(* CODESYS project ExampleProject 1.0.0.0.project

Project tree, tasks and I/O mapping:
  CODESYS_Control_for_Raspberry_Pi_SL : CODESYS Control for Raspberry Pi SL, 3S - Smart Software Solutions GmbH, version 3.5.12.0
    application Application
      libraries: Util, * (System)
      task Task (cyclic, interval t#50ms, priority 1, watchdog 100 ms x 1) calls PRG_Monarco_HAT_Examples
      task VISU_TASK (cyclic, interval 100 ms, priority 31) calls VisuElems.Visu_Prg
      program PRG_Monarco_HAT_Examples [ST]
      RS485/
        Enums/
          data type SERIAL_LINE_MODE
        FB/
          function block SERIAL_LINE [ST]: Fb_init, CLOSE
        Visualisation/
          visualisation Visualisation
          visualisation SERIAL_LINE_VISU
    SoftMotion General Axis Pool
    I²C
    SPI
      SPI_master : SPI master, 3S - Smart Software Solutions GmbH, version 1.0.0.0
          settings: _diBitsPerWord = 8; _diMaxSpeed = 1000000
        Monarco_HAT : Monarco HAT, Monarco.io, version 1.0.0.0
    GPIOs_A_B : GPIOs B+/Pi2, 3S - Smart Software Solutions GmbH, version 3.5.11.0
        unmapped channels: digital inputs (GPIO0..GPIO31), digital outputs (GPIO0..GPIO31)
    Onewire
    Camera device
      <Empty>
  libraries: Raspberry Pi Peripherals, 3.5.11.0 (3S - Smart Software Solutions GmbH); IoStandard, * (System); CAA Types Extern, * (CAA Technical Workgroup); Standard, * (System); SysTypes Interfaces, * (System); CAA Memory, * (CAA Technical Workgroup); Component Manager, * (System); CmpLog, * (System); CmpErrors Interfaces, * (System); CAA SerialCom, * (CAA Technical Workgroup); CAA Real Time Clock Extern, * (CAA Technical Workgroup); VisuSymbols, 3.5.10.0 (System)
  text list GlobalTextList
*)

// CODESYS_Control_for_Raspberry_Pi_SL/Application/RS485/Enums/SERIAL_LINE_MODE
TYPE SERIAL_LINE_MODE : (SL_READ, SL_WRITE, SL_READWRITE);
END_TYPE

// CODESYS_Control_for_Raspberry_Pi_SL/Application/PRG_Monarco_HAT_Examples
PROGRAM PRG_Monarco_HAT_Examples
VAR
	xOPm 			: BOOL := FALSE;// is the SPI master operational?
	xOPs			: BOOL := FALSE;// is the SPI slave operational?
	xExecute		: BOOL := TRUE;
	I				: INT;
	LedValue		: BYTE;	

	uiWDTime 		: UINT := 123;
	uiNewWDTime		: UINT := 500;
	xSetWd			: BOOL := FALSE;
	xWrite			: BOOL;
	DOut			: MNR.stDOut;
	DIn				: MNR.stDIn;
	AOut			: MNR.stAOut;     		
	AIn				: MNR.stAIn;	
	K	 			: INT;
	
	HatInfo			: MNR.stHATinfo;
	
	xSetHwConfig1	: BOOL;
	xGetHwConfig1	: BOOL;
	xTerminated		: BOOL;
	xAIN1shunt		: BOOL;
	xAIN2shunt		: BOOL;
	myHWConfig1		: MNR.stHWConfig1;
	curHWConfig1	: MNR.stHWConfig1;
	
	Blink			: UTIL.BLINK;
	GetDateAndTime	: RTCLK.GetDateAndTime;
	xEnablePWM		: BOOL;
	xDone			: BOOL;
	xBusy			: BOOL;
	xError			: BOOL;
	eError			: RTCLK.ERROR;
	eTimezone		: RTCLK.PERIODE;
	VarTimeCur		: DATE_AND_TIME;
	
	xSetConfig		: BOOL;
	xGetConfig		: BOOL;
	eMode			: MNR.eCounterMode 			:= MNR.eCounterMode.Off;
	eDirection		: MNR.eCounterDirection 	:= MNR.eCounterDirection.Up;
	eActiveEdge		: MNR.eCounterActiveEdge	:= MNR.eCounterActiveEdge.Rising;
	eCapture		: MNR.eCounterCapture		:= MNR.eCounterCapture.Disabled;
	myConfig1 		: MNR.stCounter1Config;
	getConfig1		: MNR.stCounter1Config;
	
	xTwoLinesOld	: BOOL;
	FirstSerialLine	: SERIAL_LINE;	
	uiCurBaudrate	: UINT;	
	xGetBaudrate	: BOOL := TRUE;
	xSetBaudrate	: BOOL;           	
	xSetMode		: BOOL;
	xGetMode		: BOOL;
	xSetRS485Mode	: BOOL;
	xGetRS485Mode	: BOOL;
	eDatabits		: MNR.eRS485Databits 	:= MNR.eRS485Databits.eight;
	eParity			: MNR.eRS485Parity 		:= MNR.eRS485Parity.none;
	eStopbits		: MNR.eRS485Stopbits 	:= MNR.eRS485Stopbits.One;
	ServiceResponse : MNR.stServiceResponse;
	myMode 			: MNR.stRS485Mode;
	xGetHOSTBaudrate: BOOL := TRUE;
	uiHOSTBaudrate	: UINT;
END_VAR

(*============================== VARIOUS HAT DEMONSTRATION USAGE EXAMPLES ==============================
	Wiring for Monarco self test;
	Wire all AO channels to the AI channels (2 AO, 2 AI),
	Wire all DO channels to the DI channels (4 DO, 4 DI),
	Wire the GND to DIn COM-,
	Wire RS485 Rx to Tx,
	Ready!
*)
xOPm  := SPI_Master.Operational;
xOPs  := Monarco_HAT.Operational;
HatInfo	:= Monarco_HAT.HATinfo;


(*============================== Monarco Leds  ==============================*)
IF I <= 7 THEN
	I := I + 1;
ELSE
	I := 0;
END_IF
LEDValue 			:= TO_BYTE( EXPT(2,I) );
Monarco_HAT.SetUserLED( byLeds := LEDValue);


(*============================== Watchdog  ==============================*)
uiWDTime    := Monarco_HAT.Watchdog;
IF xSetWd THEN
	// set
	Monarco_HAT.Watchdog := uiNewWDTime;
	xSetWd	:= FALSE;
END_IF


(*============================== Monarco DO as a struct  ==============================*)
K := K + 1;
IF K > 4 THEN
	K := 0;
END_IF;
DOut.xDOut1 := (K=1);
DOut.xDOut2 := (K=2);
DOut.xDOut3 := (K=3);
DOut.xDOut4 := (K=4);
Monarco_HAT.setDOut( stDOut := Dout);
/// two "overloads" are available;
//Monarco_HAT.setDOutBool 
//Monarco_HAT.setDOutByte

(*============================== Monarco DI as a struct  ==============================*)
Monarco_HAT.getDIn( stDIn => DIn );
///two "overloads" are available;
//Monarco_HAT.getDInBool
//Monarco_HAT.getDInByte


(*============================== Monarco AO as a struct  ==============================*)
AOut.wAOut1 := AOut.wAOut1 + 1;
IF AOut.wAOut1 >4095 THEN
	AOut.wAOut1 := 0;
END_IF
AOut.wAOut2 := AOut.wAOut1;
Monarco_HAT.setAOut( stAOut := AOut );
/// One "overload" is available;
//Monarco_Hat.setAOutWord


(*============================== AI as a struct  ==============================*)
Monarco_HAT.getAIn( stAIn => AIn);
/// One "overload" is available;
//Monarco_Hat.getAInWord


(*============================== HWCONFIG ==============================*)
// read current config
IF xGetHwConfig1 THEN
	curHWConfig1 := Monarco_HAT.HWConfig1;
	xGetHwConfig1 := FALSE;
END_IF

IF xSetHwConfig1 THEN
	myHWConfig1.xTerminated := xTerminated;
	myHWConfig1.xAIn1shunt  := xAIN1shunt;
	myHWConfig1.xAIN2shunt  := xAIN2shunt;
	// set new config
	Monarco_HAT.HWConfig1 := myHWConfig1;
	// read current config
	xGetHwConfig1 := TRUE;
	xSetHwConfig1 := FALSE;
END_IF


(*============================== One Wire ==============================*)
// One Wire is ready to use after the HAT overlay is installed
// A usage example is not provided

(*============================== RTC ==============================*)
// RTC is ready to use after the HAT overlay is installed
Blink( ENABLE := TRUE, TIMELOW := T#500MS, TIMEHIGH := T#500MS);
GetDateAndTime(
	xExecute:= Blink.OUT, // pulse for actual time
	xDone=> xDone, 
	xBusy=> xBusy, 
	xError=> xError, 
	eError=> eError, 
	eTimezone=> eTimezone);
IF xDone AND NOT xError THEN
	VarTimeCur := GetDateAndTime.dtDateAndTime;
END_IF


(*============================== COUNTER ==============================*)
// Setting an arbitrairy mode via property
myConfig1.eMode			:= eMode;
myConfig1.eDirection	:= eDirection;
myConfig1.eActiveEdge	:= eActiveEdge;
IF xSetConfig THEN
	Monarco_HAT.Counter1Config := myConfig1;
	xSetConfig := FALSE;
END_IF
IF xGetConfig THEN
	getConfig1 := Monarco_HAT.Counter1Config;
	xGetConfig := FALSE;
END_IF


(*============================== PWM ==============================*)
Monarco_HAT.setPWM1freq( udiHz := 5000); // 5000Hz
Monarco_HAT.setPWM2freq( udiHz := 100); // 100Hz
IF xEnablePWM THEN
	Monarco_HAT.setDutyCycleDOut1(rDutyCycle := 0.04); //4%
	Monarco_HAT.setDutyCycleDOut2(rDutyCycle := 0.20); //20%
	Monarco_HAT.setDutyCycleDOut3(rDutyCycle := 0.45); //45%
	Monarco_HAT.setDutyCycleDOut4(rDutyCycle := 0.75); //75%
ELSE
	/// Disable the PWM
	Monarco_HAT.setDutyCycleDOut1(rDutyCycle := 0.0); //0%
	Monarco_HAT.setDutyCycleDOut2(rDutyCycle := 0.0); //0%
	Monarco_HAT.setDutyCycleDOut3(rDutyCycle := 0.0); //0%
	Monarco_HAT.setDutyCycleDOut4(rDutyCycle := 0.0); //0%
END_IF


(*============================== Counters ==============================*)
// Counters are ready to use after the HAT overlay is installed
// A usage example is not provided


(*============================== RS485 ==============================*)
//// Adapt the enums for COM library interoperability, in this case Monarco.IO to CAA_COM_LIB;
//CASE getMode.Databits OF
//	MNR.eRS485Databits.Five			: udiByteSize := 5;
//	MNR.eRS485Databits.Six			: udiByteSize := 6;
//	MNR.eRS485Databits.Seven		: udiByteSize := 7;
//	MNR.eRS485Databits.Eight		: udiByteSize := 8;
//END_CASE
//CASE getMode.Parity OF
//	MNR.eRS485Parity.Even			: paParity := COM.PARITY.EVEN;
//	MNR.eRS485Parity.Odd			: paParity := COM.PARITY.ODD;
//	MNR.eRS485Parity.None			: paParity := COM.PARITY.None;
//END_CASE
//CASE getMode.Stopbits OF
//	MNR.eRS485STOPBITS.One			: sbStopBits := COM.STOPBIT.ONESTOPBIT;	
//	MNR.eRS485STOPBITS.OneAndAHalf	: sbStopBits := COM.STOPBIT.ONE5STOPBITS;	
//	MNR.eRS485STOPBITS.Two			: sbStopBits := COM.STOPBIT.TWOSTOPBITS;
//ELSE
//// 1/2 stopbit *not* supported in CAA COM lib!
//	MNR.eRS485STOPBITS.Half			: sbStopBits := COM.STOPBIT.ONESTOPBIT;
//END_CASE

IF xGetBaudrate THEN
	uiCurBaudrate := Monarco_HAT.RS485Baudrate;
	xGetBaudrate := FALSE;
END_IF
IF xSetBaudrate THEN
	// set 320000 baud 
	Monarco_HAT.RS485Baudrate := 320;
	xSetBaudrate := FALSE;
END_IF
// Setting the mode via a service request
IF xSetMode THEN
	// Setting 8,E,1 (Default 8,N,1)
	Monarco_HAT.serviceRequest( wValue := 16#0039, eCommand := MNR.eServiceCommand.SDC_FIXED_RS485MODE, xWrite := TRUE);
	xSetMode := FALSE;
END_IF
// Reading HOST UART mode via a service request
IF xGetMode THEN
	Monarco_HAT.serviceRequest( wValue := MNR.ParamList.MONARCO_SERVICE_STATUS_OK, eCommand := MNR.eServiceCommand.SDC_FIXED_HOST_UART, xWrite := FALSE);
	xGetMode := FALSE;
	// Read last response, default will be 16#0038 (8,N,1)
	// When setmode this will yield 16#0039
	Monarco_HAT.getServiceResponse(Response => ServiceResponse);
END_IF
// Setting an arbitrairy mode via property
myMode.eDatabits	:= eDatabits;
myMode.eParity		:= eParity;
myMode.eStopbits	:= eStopbits;
IF xSetRS485Mode THEN
	Monarco_HAT.RS485Mode := myMode;
	xSetRS485Mode := FALSE;
END_IF
IF xGetRS485Mode THEN
	myMode := Monarco_HAT.RS485Mode;
	xGetRS485Mode := FALSE;
END_IF
// should be 115200
IF xGetHOSTBaudrate THEN
 	uiHostBaudrate := Monarco_HAT.HostBaudrate;
	xGetHOSTBaudrate := FALSE;
END_IF;

// Sourcecode is included in this project under a separate RS485 section
FirstSerialLine(
		slMode:= SL_READWRITE, 
		udiPort:= 1, 							
		udiBaudrate:= 115200,
		paParity:= COM.PARITY.NONE,
		sbStopBits:= COM.STOPBIT.ONESTOPBIT,
		udiByteSize := 8);

END_PROGRAM

// CODESYS_Control_for_Raspberry_Pi_SL/Application/RS485/FB/SERIAL_LINE
FUNCTION_BLOCK SERIAL_LINE
VAR_INPUT
	slMode				: SERIAL_LINE_MODE;
	udiPort				: UDINT;
	udiBaudrate			: UDINT;
	sbStopBits			: COM.STOPBIT:= COM.STOPBIT.ONESTOPBIT;
	paParity			: COM.PARITY:= COM.PARITY.EVEN;
	sWriteText			: STRING:= 'Hello Raspberry and Monarco! ';
	udiByteSize			: UDINT;
END_VAR
VAR_OUTPUT
	sReadText			: STRING;
	errError			: COM.ERROR;
	xReadSuccess		: BOOL;
	xWriteSuccess		: BOOL;
	xClosed				: BOOL:= TRUE;
END_VAR
VAR
	iState				: INT;
	tTimer				: TON;
	comOpen				: COM.Open; (* Instance of the function block for opening a port *)
	hCom				: CAA.HANDLE; (* handle of the port*)
	aParameter			: ARRAY [1..7] OF COM.PARAMETER;
	comWrite			: COM.Write;	(* Instance of the Write function  block *)
	bWriteBuffer		: ARRAY [1..80] OF BYTE; (*Used to write data to the serial port*)
	szWrite				: CAA.SIZE;
	comRead				: COM.Read; (* Instance of the Read function block *)
	bReadBuffer			: ARRAY [1..80] OF BYTE; (*Used to read data from the serial port*)
	szRead				: CAA.SIZE;
	comClose			: COM.Close; (* Instance of the function block for closing a port *)
END_VAR

CASE iState OF
	
	0:	// The parameter for the COM Ports are set
		aParameter[1].udiParameterId:= COM.CAA_Parameter_Constants.udiPort;
		aParameter[1].udiValue:= udiPort;
		aParameter[2].udiParameterId:= COM.CAA_Parameter_Constants.udiBaudrate;
		aParameter[2].udiValue:= udiBaudrate;		
		aParameter[3].udiParameterId:= COM.CAA_Parameter_Constants.udiStopBits;
		aParameter[3].udiValue:= sbStopBits;
		aParameter[4].udiParameterId:= COM.CAA_Parameter_Constants.udiParity;
		aParameter[4].udiValue:= paParity;
		aParameter[5].udiParameterId:= COM.CAA_Parameter_Constants.udiTimeout;
		aParameter[5].udiValue:= 0;
		aParameter[6].udiParameterId:= COM.CAA_Parameter_Constants.udiBinary;
		aParameter[6].udiValue:= 0;
		aParameter[7].udiParameterId:= COM.CAA_Parameter_Constants.udiByteSize;
		aParameter[7].udiValue:= udiByteSize;
		
		iState:= 1;
		
	1:	//First the COM Port is opened
		comOpen(xExecute:= TRUE, usiListLength:= SIZEOF(aParameter) / SIZEOF(COM.PARAMETER), pParameterList:= ADR(aParameter), hCom=> hCom);
		xClosed:= FALSE;
		IF comOpen.xDone THEN
			comOpen(xExecute:= FALSE);
			//depending on the mode the state for reading or writing is set
			IF slMode = SL_READ OR slMode = SL_READWRITE THEN
				iState:= 2;
			ELSIF slMode = SL_WRITE THEN
				iState:= 4;
			END_IF
		ELSIF comOpen.xError THEN
			errError:= comOpen.eError;
			comOpen(xExecute:= FALSE);
			iState:= 32767;
		END_IF
		
	2: //The reading process is started
		comRead(xExecute:= TRUE, hCom:= hCom, pBuffer:= ADR(bReadBuffer), szBuffer:= SIZEOF(bReadBuffer));
		IF comRead.xDone THEN
			szRead:= comRead.szSize;
			//check if the Port has send something
			IF szRead > 0 THEN
				//the text from the read buffer is saved in the sReadText variable
				MEM.MemMove(ADR(bReadBuffer), ADR(sReadText), UDINT_TO_UINT(szRead));
				MEM.MemFill(ADR(sReadText) + UDINT_TO_UINT(szRead), 1, 0);
				xReadSuccess:= TRUE;
			END_IF
			// the flag has to be set to false, that in the next cylce, the read task will start again, by setting it to true
			comRead(xExecute:= FALSE);
			iState:= 3;
		ELSIF comRead.xError THEN
			errError:= comRead.eError;
			comRead(xExecute:= FALSE);
			iState:= 32767;
		END_IF
		
	3: //After the reading process is finished, a timer is started for waiting 250 milliseconds
		tTimer(IN:= TRUE, PT:= T#250MS);
		IF tTimer.Q THEN
			tTimer(IN:= FALSE);
			xReadSuccess:= FALSE;
			IF slMode = SL_READWRITE THEN
				iState:= 4;
			ELSE
				iState:= 2;
			END_IF
		END_IF
		
	4: // the writing process is started
		IF NOT comWrite.xExecute THEN
			szWrite:= INT_TO_UDINT(LEN(sWriteText));
			//write the string to the buffer for the COM.WRITE Interface
			MEM.MemMove(ADR(sWriteText), ADR(bWriteBuffer), UDINT_TO_UINT(szWrite));
		END_IF
		comWrite(xExecute:= TRUE, hCom:= hCom, pBuffer:= ADR(bWriteBuffer), szSize:= szWrite);
		IF comWrite.xDone THEN
			// the flag is set to false, that in the next cyle this process is started again, by setting it to true 
			comWrite(xExecute:= FALSE);	
			xWriteSuccess:= TRUE;
			iState:= 5;
		ELSIF comWrite.xError THEN
			errError:= comWrite.eError;
			comWrite(xExecute:= FALSE);	
			iState:= 32767;
		END_IF 
		
	5: //After the writing process is finished, a timer is started for waiting 250 milliseconds
		tTimer(IN:= TRUE, PT:= T#250MS);
		IF tTimer.Q THEN
			tTimer(IN:= FALSE);
			xWriteSuccess:= FALSE;
			IF slMode = SL_READWRITE THEN
				iState:= 2;
			ELSE
				iState:= 4;
			END_IF
		END_IF
		
	6: //Closing the ports
		IF hCom <> 0 THEN
			comClose(xExecute:= TRUE, hCom:= hCom);
			IF comClose.xDone THEN
				comClose(xExecute:= FALSE);
				Fb_Init(FALSE, FALSE);
			ELSIF comClose.xError THEN
				errError:= comClose.eError;
				comClose(xExecute:= FALSE);	
				iState:= 32767;
			END_IF
		ELSE
			Fb_Init(FALSE, FALSE);
		END_IF 

	32767:
		;

END_CASE

METHOD Fb_init : BOOL
VAR_INPUT
	bInitRetains : BOOL;
  	bInCopyCode : BOOL; 
END_VAR
END_METHOD

ACTION CLOSE:
iState:= 6;
THIS^();
END_ACTION

END_FUNCTION_BLOCK

// CODESYS_Control_for_Raspberry_Pi_SL/Application/RS485/Visualisation/Visualisation
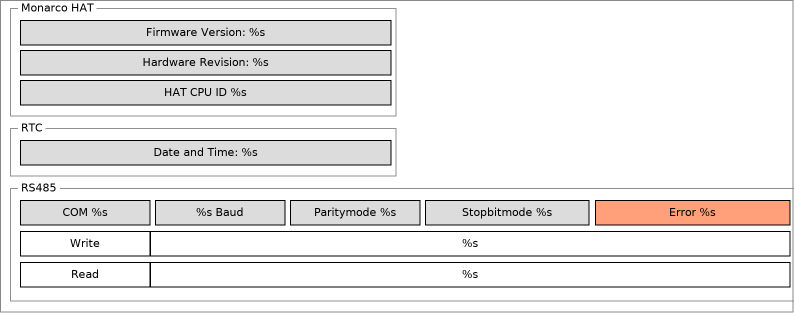
VISUALIZATION Visualisation  // 794x313
    Frame (5,180 787x131)
        shows SERIAL_LINE_VISU(slInstance := PRG_Monarco_HAT_Examples.FirstSerialLine)
    GroupBox (10,0 386x116), "Monarco HAT"
        Rectangle (10,20 371x25), "Firmware Version: %s", text variable: PRG_Monarco_HAT_Examples.HATinfo.dwFwVersion
        Rectangle (10,50 371x25), "Hardware Revision: %s", text variable: PRG_Monarco_HAT_Examples.HATinfo.dwHwversion
        Rectangle (10,80 371x25), "HAT CPU ID %s", text variable: PRG_Monarco_HAT_Examples.HATinfo.lwCpuID
    GroupBox (10,120 386x56), "RTC"
        Rectangle (10,20 371x25), "Date and Time: %s", text variable: PRG_Monarco_HAT_Examples.VarTimeCur
END_VISUALIZATION

// CODESYS_Control_for_Raspberry_Pi_SL/Application/RS485/Visualisation/SERIAL_LINE_VISU
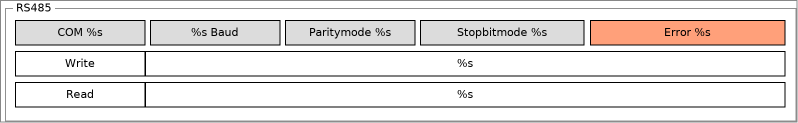
VISUALIZATION SERIAL_LINE_VISU  // 798x123
VAR_IN_OUT
	slInstance: SERIAL_LINE;
END_VAR
    GroupBox (5,0 791x121), "RS485"
        Rectangle (140,51 640x25), "%s", text variable: slInstance.sWriteText, invisible if: slInstance.slMode = SL_READ
            OnMouseDown: write the text variable via Edit
        Rectangle (10,51 130x25), "Write", colour toggle: slInstance.xWriteSuccess, invisible if: slInstance.slMode = SL_READ
        Rectangle (140,82 640x25), "%s", text variable: slInstance.sReadText, invisible if: slInstance.slMode = SL_WRITE
        Rectangle (10,82 130x25), "Read", colour toggle: slInstance.xReadSuccess, invisible if: slInstance.slMode = SL_WRITE
        Rectangle (10,20 130x25), "COM %s", text variable: slInstance.udiPort
        Rectangle (145,20 130x25), "%s Baud", text variable: slINstance.udiBaudrate
        Rectangle (585,20 195x25), "Error %s", text variable: slInstance.errError
        Rectangle (280,20 130x25), "Paritymode %s", text variable: slInstance.paParity
        Rectangle (415,20 164x25), "Stopbitmode %s", text variable: slInstance.sbStopBits
END_VISUALIZATION
